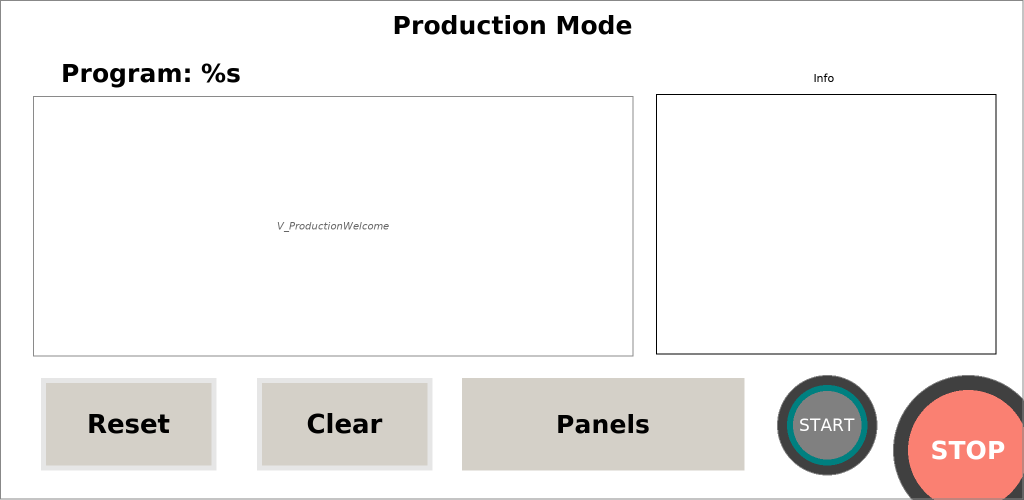
VISUALIZATION V_ProductionMode  // 1024x500
VAR_IN_OUT
	HMI : ST_PackMLBaseModule_HMI;
	HMI_GantryXYZ : ST_GantryXYZ_HMI;
	HMI_Recipe : ST_RecipeBuilder_HMI;
END_VAR
    Label (0,0 1025x50), "Production Mode"
    RoundedRectangle (257,378 175x92), "Clear", colour toggle: (HMI.Status.State = E_PMLState.ePMLState_Aborted) OR (HMI.Status.State = E_PMLState.ePMLState_Clearing)
        OnMouseClick: execute { HMI.Command.State := E_PMLCommand.ePMLCommand_Clear; }
    RoundedRectangle (41,378 175x92), "Reset", colour toggle: (HMI.Status.State = E_PMLState.ePMLState_Complete) OR (HMI.Status.State = E_PMLState.ePMLState_Stopped) OR (HMI.Status.State = E_PMLState.ePMLState_Resetting)
        OnMouseClick: execute { HMI.Command.State := E_PMLCommand.ePMLCommand_Reset; }
    Frame (33,96 600x260), frame switch variable: HMI_GantryXYZ.Command.ProgramIdRequested
        shows V_ProductionWelcome()
        shows V_ProductionBorgoFlaps(HMI := MAIN.Seedra.PackMLBaseModule_HMI, HMI_GantryXYZ := MAIN.Seedra.GantryXYZ.GantryXYZ_HMI, HMI_Recipe := MAIN.Seedra.RecipeConfig_HMI)
        shows V_ProductionBorgoWings(HMI := MAIN.Seedra.PackMLBaseModule_HMI, HMI_GantryXYZ := MAIN.Seedra.GantryXYZ.GantryXYZ_HMI, HMI_Recipe := MAIN.Seedra.RecipeConfig_HMI)
        shows V_ProductionArona(HMI := MAIN.Seedra.PackMLBaseModule_HMI, HMI_GantryXYZ := MAIN.Seedra.GantryXYZ.GantryXYZ_HMI, HMI_Recipe := MAIN.Seedra.RecipeConfig_HMI)
        shows V_ProductionNCICircle(HMI := MAIN.Seedra.PackMLBaseModule_HMI, HMI_GantryXYZ := MAIN.Seedra.GantryXYZ.GantryXYZ_HMI, HMI_Recipe := MAIN.Seedra.RecipeConfig_HMI)
        shows V_ProductionRectangle(HMI := MAIN.Seedra.PackMLBaseModule_HMI, HMI_GantryXYZ := MAIN.Seedra.GantryXYZ.GantryXYZ_HMI, HMI_Recipe := MAIN.Seedra.RecipeConfig_HMI)
        shows V_ProductionRoundRectangle(HMI := MAIN.Seedra.PackMLBaseModule_HMI, HMI_GantryXYZ := MAIN.Seedra.GantryXYZ.GantryXYZ_HMI, HMI_Recipe := MAIN.Seedra.RecipeConfig_HMI)
        shows V_ProductionFeedCircle(HMI := MAIN.Seedra.PackMLBaseModule_HMI, HMI_GantryXYZ := MAIN.Seedra.GantryXYZ.GantryXYZ_HMI, HMI_Recipe := MAIN.Seedra.RecipeConfig_HMI)
        shows V_Meina2_2000x1000(HMI := MAIN.Seedra.PackMLBaseModule_HMI, HMI_GantryXYZ := MAIN.Seedra.GantryXYZ.GantryXYZ_HMI, HMI_Recipe := MAIN.Seedra.RecipeConfig_HMI)
        shows V_ProductionMeina2_5Squares(HMI := MAIN.Seedra.PackMLBaseModule_HMI, HMI_GantryXYZ := MAIN.Seedra.GantryXYZ.GantryXYZ_HMI, HMI_Recipe := MAIN.Seedra.RecipeConfig_HMI)
        shows V_ProductionMeina2_5Circles(HMI := MAIN.Seedra.PackMLBaseModule_HMI, HMI_GantryXYZ := MAIN.Seedra.GantryXYZ.GantryXYZ_HMI, HMI_Recipe := MAIN.Seedra.RecipeConfig_HMI)
        shows V_ProductionMeina2_3Squares(HMI := MAIN.Seedra.PackMLBaseModule_HMI, HMI_GantryXYZ := MAIN.Seedra.GantryXYZ.GantryXYZ_HMI, HMI_Recipe := MAIN.Seedra.RecipeConfig_HMI)
        shows V_ProductionMeina2_3Circles(HMI := MAIN.Seedra.PackMLBaseModule_HMI, HMI_GantryXYZ := MAIN.Seedra.GantryXYZ.GantryXYZ_HMI, HMI_Recipe := MAIN.Seedra.RecipeConfig_HMI)
        shows V_ProductionMeina2_2Squares(HMI := MAIN.Seedra.PackMLBaseModule_HMI, HMI_GantryXYZ := MAIN.Seedra.GantryXYZ.GantryXYZ_HMI, HMI_Recipe := MAIN.Seedra.RecipeConfig_HMI)
        shows V_ProductionMeina2_2Circles(HMI := MAIN.Seedra.PackMLBaseModule_HMI, HMI_GantryXYZ := MAIN.Seedra.GantryXYZ.GantryXYZ_HMI, HMI_Recipe := MAIN.Seedra.RecipeConfig_HMI)
        shows V_ProductionMeina2_2Rectangles(HMI := MAIN.Seedra.PackMLBaseModule_HMI, HMI_GantryXYZ := MAIN.Seedra.GantryXYZ.GantryXYZ_HMI, HMI_Recipe := MAIN.Seedra.RecipeConfig_HMI)
        shows V_Meina2_Samples(HMI := MAIN.Seedra.PackMLBaseModule_HMI, HMI_GantryXYZ := MAIN.Seedra.GantryXYZ.GantryXYZ_HMI, HMI_Recipe := MAIN.Seedra.RecipeConfig_HMI)
        p3843536458: MAIN.Seedra.RecipeBuilderWings.RecipeBuilder_HMI
    RoundedRectangle (656,94 340x260)
    Group (893,375 100x100)
        Ellipse (0,0 150x150)
        Ellipse (15,15 120x120), "STOP"
            toggle GVL_Safety.eStopHMI
    Label (679,66 290x25), "Info"
    RoundedRectangle (462,378 282x92), "Panels"
        OnMouseClick: execute { GVL_HMI.PopupToDisplay := 2; }
    Textfield (58,57 531x32), "Program: %s", text variable: MAIN.Seedra.sSelectedRecipeName
    Ellipse (777,375 100x100)
    Ellipse (787,385 80x80), "START", colour toggle: HMI.Status.State = E_PMLState.ePMLState_Idle, input disabled if: NOT MAIN.Seedra.RecipeConfig_HMI.Config.IsValid
        OnMouseClick: execute { HMI.Command.State := E_PMLCommand.ePMLCommand_Start; }
END_VISUALIZATION

(* stored: Version 1.1.0.1, ProductVersion 3.1.4024.15
   Visu V_ProductionMode: Id {36f6a3ae-b99e-0ef0-3759-f9efb58a3c39} *)
